Staubli VAL3: recvIoWriteRequest.pgx

public program recvIoWriteRequest(bool& x_bFlag)
begin
  // Copyright (c) 2016, Ocado Technology - Robotics Research Team
  //
  // Licensed under the Apache License, Version 2.0 (the "License");
  // you may not use this file except in compliance with the License.
  // You may obtain a copy of the License at
  //
  //     http://www.apache.org/licenses/LICENSE-2.0
  //
  // Unless required by applicable law or agreed to in writing, software
  // distributed under the License is distributed on an "AS IS" BASIS,
  // WITHOUT WARRANTIES OR CONDITIONS OF ANY KIND, either express or implied.
  // See the License for the specific language governing permissions and
  // limitations under the License.



  // attempt to receive message ID 65202 data (prefix and header are in rosGenericMsg)
  rosIoWriteRequestMsg.prefix.nLength=rosGenericMsg.prefix.nLength
  rosIoWriteRequestMsg.header.nMsgType=rosGenericMsg.header.nMsgType
  rosIoWriteRequestMsg.header.nCommType=rosGenericMsg.header.nCommType
  rosIoWriteRequestMsg.header.nReplyCode=rosGenericMsg.header.nReplyCode

  call recvData(siTcpIpMotion,rosIoWriteRequestMsg.body.nData,nInConnFlag,x_bFlag)
end
